FUNCTION_BLOCK DataPanel_MI_IW_0_10V (* Input service interface function block for analog input data (0-10V) *)
  (* Description: Copyright (c) 2026 HR Agrartechnik GmbH *)
  (* Version 1.0, 2026-01-17, generated, HR Agrartechnik GmbH *)
  PACKAGE DataPanel::io::MI::AI;
  IMPORT DataPanel::io::MI::const::MI;
  IMPORT eclipse4diac::core::TypeHash;
  IMPORT DataPanel::io::MI::AI::DataPanel_MI_AI::Invalid;
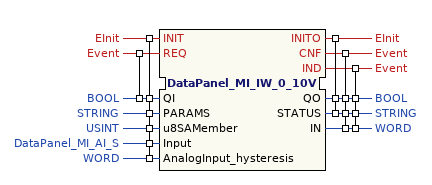
  EVENT_INPUT
    INIT : EInit WITH QI, PARAMS, u8SAMember, Input, AnalogInput_hysteresis; (* Service Initialization *)
    REQ WITH QI; (* Service Request *)
  END_EVENT
  EVENT_OUTPUT
    INITO : EInit WITH QO, STATUS; (* Initialization Confirm *)
    CNF WITH QO, STATUS, IN; (* Confirmation of Requested Service *)
    IND WITH QO, STATUS, IN; (* Indication from Resource *)
  END_EVENT
  VAR_INPUT
    QI : BOOL; (* Event Input Qualifier *)
    PARAMS : STRING; (* Service Parameters *)
    u8SAMember : USINT := MI::MI_00; (* Node SA 224..239 *)
    Input : DataPanel::io::MI::AI::DataPanel_MI_AI_S := Invalid; (* Identify the Input AnalogInput_1A..8B *)
    AnalogInput_hysteresis : WORD;
  END_VAR
  VAR_OUTPUT
    QO : BOOL; (* Event Output Qualifier *)
    STATUS : STRING; (* Service Status *)
    IN : WORD; (* Input data from resource *)
  END_VAR
END_FUNCTION_BLOCK
